FUNCTION_BLOCK CNV_TRANSFER (* Composite Function Block Type *)
  (* Standard: 61499-2 *)
  (* Version 0.2, 2003-12-05, JHC, Rockwell Automation, Renamed from NEWCOMPFB. *)
  (* Version 0.1, 2002-01-08, JHC, Rockwell Automation, Added DLY FB as example. *)
  (* Version 0.0, 2000-05-27, JHC, Rockwell Automation *)
  (* Compiler header: package fb.rt.student; *)
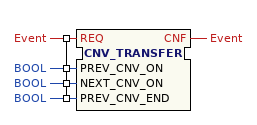
  EVENT_INPUT
    REQ WITH PREV_CNV_ON, NEXT_CNV_ON, PREV_CNV_END; (* Normal Execution Request *)
  END_EVENT
  EVENT_OUTPUT
    CNF; (* Execution Confirmation *)
  END_EVENT
  VAR_INPUT
    PREV_CNV_ON : BOOL;
    NEXT_CNV_ON : BOOL;
    PREV_CNV_END : BOOL;
  END_VAR
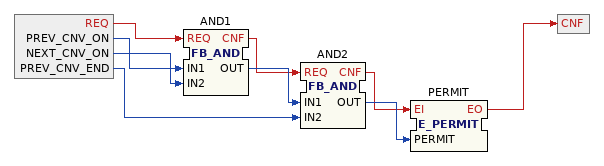
  FBS
    AND1 : FB_AND;
    AND2 : FB_AND;
    PERMIT : E_PERMIT;
  END_FBS
  EVENT_CONNECTIONS
    AND1.CNF TO AND2.REQ;
    REQ TO AND1.REQ;
    AND2.CNF TO PERMIT.EI;
    PERMIT.EO TO CNF;
  END_CONNECTIONS
  DATA_CONNECTIONS
    AND1.OUT TO AND2.IN1;
    PREV_CNV_ON TO AND1.IN1;
    NEXT_CNV_ON TO AND1.IN2;
    PREV_CNV_END TO AND2.IN2;
    AND2.OUT TO PERMIT.PERMIT;
  END_CONNECTIONS
END_FUNCTION_BLOCK
